PROGRAM analogSignals_ex02_1
VAR
	Frawsensor			: REAL;
	potentiometervalue	: REAL;
	
	LIN_TRAFO 			: FB_Scale;
END_VAR

LIN_TRAFO(
	fIN:= frawsensor, 
	fIN_min:= 0, 
	fIN_max:= 20, 
	fOUT_min:= 0, 
	fOUT_max:= 60, 
	fOUT=> potentiometervalue);

END_PROGRAM

(* stored: Version 1.1.0.1
   POU analogSignals_ex02_1: Id {2389053f-b0ea-466c-abbb-a044e0555fc9}, SpecialFunc None *)
